// TIA Portal V18 export
TYPE "PLCtoMES_ST350"
// stored: IsFailsafeCompliant false
   STRUCT
      Common { S7_SetPoint := 'True'} : "PLCtoMES_Common";   // PLC发送公共交互数据到MES
      MainCheckIn { S7_SetPoint := 'True'} : "PLCtoMES_MainCheckIn";   // PLC发送主件请求交互数据到MES
      SubCheckIn { S7_SetPoint := 'True'} : "PLCtoMES_SubCheckIn";   // PLC发送子零件绑定交互数据到MES
      Processing { S7_SetPoint := 'True'} : "PLCtoMES_ProcessingExchange";   // PLC发送Processing请求,表明工件已经入不可逆工艺,比如压装工位等
      MainCheckOut { S7_SetPoint := 'True'} : "PLCtoMES_MainCheckOut";   // PLC发送保存请求到MES
      PrintExchange { S7_SetPoint := 'True'} : "PLCtoMES_PrintExchange";   // PLC发送打印交互数据到MES
      AGVExchange { S7_SetPoint := 'True'} : "PLCtoMES_AGVExchange";   // PLC发送AGV交互数据到MES
      ProcessData { S7_SetPoint := 'True'} : "PLCtoMES_MainCheckOutProcessData_OP220";   // PLC发送结果数据到MES
      AlarmExchange { S7_SetPoint := 'True'} : "PLCtoMES_AlarmExchange";   // PLC发送设备报警数据到MES
      RealTimeData { S7_SetPoint := 'True'} : "PLCtoMES_RealTimeData";   // PLC发送实时数据到MES,MES实时读取工艺过程数据区
   END_STRUCT;
END_TYPE
